(* Calculates the size of this message in Protocol Buffer wire format, in bytes. *)
METHOD CalculateSize : UDINT
VAR
    nSize : UDINT;
    nRepeatedFieldSize : UDINT;
END_VAR
// repeated EnumOfTypeSint enum_values_sint = 1;
_fbRepeatedId1.CalculateSize(nSize => nRepeatedFieldSize);
nSize := nSize + nRepeatedFieldSize;
CalculateSize := nSize;
END_METHOD

(* Merges the data from the specified coded input stream with the current message.*)
METHOD MergeFrom : HRESULT
VAR_IN_OUT
    fbParseCtx : FB_ParseContext;
END_VAR
VAR
    nTag : UDINT;
END_VAR
_fbRepeatedId1.Initialize();
REPEAT
MergeFrom := fbParseCtx.ReadTag(nTag=> nTag);
IF SUCCEEDED(MergeFrom) AND nTag = 0 THEN
    EXIT;
END_IF;

IF FAILED(MergeFrom) THEN
    RETURN;
END_IF

CASE nTag OF
    16#0A:    // repeated EnumOfTypeSint enum_values_sint = 1;
        MergeFrom := _fbRepeatedId1.AddEntriesFrom(fbParseCtx:= fbParseCtx, ipFieldCodec:= _fbFieldCodecId1,nCount=> _stRepeatedEnumTests.enum_values_sint_count);
ELSE
    MergeFrom := fbParseCtx.SkipLastField();
END_CASE

UNTIL (FAILED(MergeFrom) OR nTag = 0)
END_REPEAT
END_METHOD

PROPERTY PUBLIC MessageValue : T_Any
GET
MessageValue := F_ToAnyType(anyArg:= _stRepeatedEnumTests);
END_GET
END_PROPERTY

PROPERTY PUBLIC Parser : REFERENCE TO FB_MessageParser
GET
Parser REF= THIS^._fbMessageParser;
END_GET
END_PROPERTY

PROPERTY PUBLIC RepeatedEnumTests : ST_RepeatedEnumTests
GET
RepeatedEnumTests := _stRepeatedEnumTests;
END_GET
SET
_stRepeatedEnumTests := RepeatedEnumTests;
END_SET
END_PROPERTY

(* Writer for this message.*)
PROPERTY PUBLIC Writer : REFERENCE TO FB_MessageWriter
GET
Writer REF= THIS^._fbMessageWriter;
END_GET
END_PROPERTY

(* Writes the data to the given coded output stream.*)
METHOD WriteTo : HRESULT
VAR_IN_OUT
	(* Coded output stream to write the data to. *)
	fbWriteCtx	: FB_WriteContext;
END_VAR
// repeated EnumOfTypeSint enum_values_sint = 1;
WriteTo := _fbRepeatedId1.WriteToWithCount(fbWriteCtx:= fbWriteCtx, ipFieldCodec:= _fbFieldCodecId1, nCount:= _stRepeatedEnumTests.enum_values_sint_count);
IF FAILED(WriteTo) THEN
    RETURN;
END_IF
END_METHOD

END_FUNCTION_BLOCK

// ---- FieldCodec/FB_FieldCodecFloat.TcPOU
FUNCTION_BLOCK FB_FieldCodecFloat EXTENDS FB_FieldCodec
VAR_INPUT
END_VAR
VAR_OUTPUT
END_VAR
VAR
    fValue : REAL;
END_VAR

METHOD CalculatePackedDataSize : HRESULT
VAR_INPUT CONSTANT
	anyFirstElem	: T_Any;
	nLength	        : UDINT;        // items to write
END_VAR
VAR_OUTPUT
    nPackedDataSize : UDINT;
END_VAR
VAR
    anyItem         : T_ANY;
    i               : UDINT;
    fValue          : REAL;
END_VAR
anyItem := anyFirstElem;

IF nLength < 1 THEN
    nPackedDataSize := 0;
    RETURN;
END_IF

FOR i := 0  TO nLength - 1 DO
    anyItem.pValue := anyFirstElem.pValue + (i * TO_UDINT(anyFirstElem.diSize)); 
    fValue := PREAL_TO_REAL(anyItem.pValue);
    nPackedDataSize := nPackedDataSize + F_ComputeFloatSize(fValue);
END_FOR
END_METHOD

METHOD IsPackedRepeatedField : BOOL
VAR_INPUT
	nTag	: UDINT;
END_VAR
IsPackedRepeatedField := F_IsPackedRepeatedField(nTag);
END_METHOD


METHOD ValueReader : HRESULT
VAR_IN_OUT      
    stCtx : ST_ParseContext;
END_VAR
VAR_OUTPUT
	anyOut	: T_Any;
END_VAR

ValueReader := F_ParseFloat(stCtx, fValue=> fValue);
anyOut := F_ToAnyType(anyArg:= fValue);
END_METHOD

METHOD ValueWriter : HRESULT
VAR_IN_OUT
    stCtx  : ST_WriteContext;
END_VAR
VAR_INPUT
    anyIn : T_ANY;
END_VAR
VAR
    fValue  : REAL;
END_VAR

fValue := PREAL_TO_REAL(anyIn.pValue);
ValueWriter := F_WriteFloat(stCtx, fValue);
END_METHOD

END_FUNCTION_BLOCK

// ---- FieldCodec/FB_FieldCodecSint32.TcPOU
FUNCTION_BLOCK FB_FieldCodecSint32 EXTENDS FB_FieldCodec
VAR_INPUT
END_VAR
VAR_OUTPUT
END_VAR
VAR
    nValue : DINT;
END_VAR

METHOD CalculatePackedDataSize : HRESULT
VAR_INPUT CONSTANT
	anyFirstElem	: T_Any;
	nLength	        : UDINT;        // items to write
END_VAR
VAR_OUTPUT
    nPackedDataSize : UDINT;
END_VAR
VAR
    anyItem         : T_ANY;
    i               : UDINT;
    nValue          : DINT;
END_VAR
anyItem := anyFirstElem;

IF nLength < 1 THEN
    nPackedDataSize := 0;
    RETURN;
END_IF

FOR i := 0  TO nLength - 1 DO
    anyItem.pValue := anyFirstElem.pValue + (i * TO_UDINT(anyFirstElem.diSize)); 
    nValue := PDINT_TO_DINT(anyItem.pValue);
    nPackedDataSize := nPackedDataSize + F_ComputeSInt32Size(nValue);
END_FOR
END_METHOD

METHOD IsPackedRepeatedField : BOOL
VAR_INPUT
	nTag	: UDINT;
END_VAR
IsPackedRepeatedField := F_IsPackedRepeatedField(nTag);
END_METHOD


METHOD ValueReader : HRESULT
VAR_IN_OUT      
    stCtx : ST_ParseContext;
END_VAR
VAR_OUTPUT
	anyOut	: T_Any;
END_VAR
VAR
    nTmp : UDINT;
END_VAR

ValueReader := F_ParseRawVarint32(stCtx, nTmp);
IF FAILED(ValueReader) THEN
    RETURN;
END_IF
nValue := F_DecodeZigZag32(nTmp);
anyOut := F_ToAnyType(anyArg:= nValue);
END_METHOD

METHOD ValueWriter : HRESULT
VAR_IN_OUT
    stCtx  : ST_WriteContext;
END_VAR
VAR_INPUT
    anyIn : T_ANY;
END_VAR
VAR
    nValue  : DINT;
END_VAR

nValue := PDINT_TO_DINT(anyIn.pValue);
ValueWriter := F_WriteSInt32(stCtx, nValue);
END_METHOD

END_FUNCTION_BLOCK

// ---- FieldCodec/FB_FieldCodecInt64.TcPOU
FUNCTION_BLOCK FB_FieldCodecInt64 EXTENDS FB_FieldCodec
VAR_INPUT
END_VAR
VAR_OUTPUT
END_VAR
VAR
    nValue : ULINT;
END_VAR

METHOD CalculatePackedDataSize : HRESULT
VAR_INPUT CONSTANT
	anyFirstElem	: T_Any;
	nLength	        : UDINT;        // items to write
END_VAR
VAR_OUTPUT
    nPackedDataSize : UDINT;
END_VAR
VAR
    anyItem         : T_ANY;
    i               : UDINT;
    nValue          : LINT;
END_VAR
anyItem := anyFirstElem;

IF nLength < 1 THEN
    nPackedDataSize := 0;
    RETURN;
END_IF

FOR i := 0  TO nLength - 1 DO
    anyItem.pValue := anyFirstElem.pValue + (i * TO_UDINT(anyFirstElem.diSize)); 
    nValue := PLINT_TO_LINT(anyItem.pValue);
    nPackedDataSize := nPackedDataSize + F_ComputeInt64Size(nValue);
END_FOR
END_METHOD

METHOD IsPackedRepeatedField : BOOL
VAR_INPUT
	nTag	: UDINT;
END_VAR
IsPackedRepeatedField := F_IsPackedRepeatedField(nTag);
END_METHOD


METHOD ValueReader : HRESULT
VAR_IN_OUT      
    stCtx : ST_ParseContext;
END_VAR
VAR_OUTPUT
	anyOut	: T_Any;
END_VAR

ValueReader := F_ParseRawVarint64(stCtx, nValue);
anyOut := F_ToAnyType(anyArg:= nValue);
END_METHOD

METHOD ValueWriter : HRESULT
VAR_IN_OUT
    stCtx  : ST_WriteContext;
END_VAR
VAR_INPUT
    anyIn : T_ANY;
END_VAR
VAR
    nValue  : LINT;
END_VAR

nValue := PLINT_TO_LINT(anyIn.pValue);
ValueWriter := F_WriteInt64(stCtx, nValue);
END_METHOD

END_FUNCTION_BLOCK

// ---- FieldCodec/FB_FieldCodecSint64.TcPOU
FUNCTION_BLOCK FB_FieldCodecSint64 EXTENDS FB_FieldCodec
VAR_INPUT
END_VAR
VAR_OUTPUT
END_VAR
VAR
    nValue : LINT;
END_VAR

METHOD CalculatePackedDataSize : HRESULT
VAR_INPUT CONSTANT
	anyFirstElem	: T_Any;
	nLength	        : UDINT;        // items to write
END_VAR
VAR_OUTPUT
    nPackedDataSize : UDINT;
END_VAR
VAR
    anyItem         : T_ANY;
    i               : UDINT;
    nValue          : LINT;
END_VAR
anyItem := anyFirstElem;

IF nLength < 1 THEN
    nPackedDataSize := 0;
    RETURN;
END_IF

FOR i := 0  TO nLength - 1 DO
    anyItem.pValue := anyFirstElem.pValue + (i * TO_UDINT(anyFirstElem.diSize)); 
    nValue := PLINT_TO_LINT(anyItem.pValue);
    nPackedDataSize := nPackedDataSize + F_ComputeSInt64Size(nValue);
END_FOR
END_METHOD

METHOD IsPackedRepeatedField : BOOL
VAR_INPUT
	nTag	: UDINT;
END_VAR
IsPackedRepeatedField := F_IsPackedRepeatedField(nTag);
END_METHOD


METHOD ValueReader : HRESULT
VAR_IN_OUT      
    stCtx : ST_ParseContext;
END_VAR
VAR_OUTPUT
	anyOut	: T_Any;
END_VAR
VAR 
    nTmp : ULINT;
END_VAR

ValueReader := F_ParseRawVarint64(stCtx, nTmp);
IF FAILED(ValueReader) THEN
    RETURN;
END_IF
nValue := F_DecodeZigZag64(nTmp);
anyOut := F_ToAnyType(anyArg:= nValue);
END_METHOD

METHOD ValueWriter : HRESULT
VAR_IN_OUT
    stCtx  : ST_WriteContext;
END_VAR
VAR_INPUT
    anyIn : T_ANY;
END_VAR
VAR
    nValue  : LINT;
END_VAR

nValue := PLINT_TO_LINT(anyIn.pValue);
ValueWriter := F_WriteSInt64(stCtx, nValue);
END_METHOD

END_FUNCTION_BLOCK

// ---- Helper/POUs/F_ToAnyBit.TcPOU
FUNCTION F_ToAnyBit : T_AnyBit
VAR_INPUT
    anyBit	: ANY_BIT;
END_VAR

F_ToAnyBit := anyBit;

END_FUNCTION

// ---- Helper/POUs/F_ToAnyInt.TcPOU
FUNCTION F_ToAnyInt : T_AnyInt
VAR_INPUT
    anyInt	: ANY_INT;
END_VAR

F_ToAnyInt := anyInt;

END_FUNCTION

// ---- Helper/POUs/F_ToAnyNum.TcPOU
FUNCTION F_ToAnyNum : T_AnyNum
VAR_INPUT
    anyNum	: ANY_NUM;
END_VAR

F_ToAnyNum := anyNum;

END_FUNCTION

// ---- ParsingPrimitives/POUs/F_ReadStringInternal.TcPOU
// Reads a string field value from the input.
FUNCTION INTERNAL F_ReadStringInternal : HRESULT
VAR_IN_OUT      
    stCtx : ST_ParseContext;
END_VAR
VAR_INPUT
    stAnyStringOut : T_Any;   
END_VAR
VAR
    nStrLength : UDINT;
END_VAR

F_ReadStringInternal := S_OK;

F_ReadStringInternal := F_ParseLength(stCtx, nLength=> nStrLength);
IF FAILED(F_ReadStringInternal) THEN
    RETURN;
END_IF

F_ReadStringInternal := F_ReadRawString(stCtx, nStrLength, stAnyStringOut);

END_FUNCTION

// ---- POUs/ComputeSize/F_ComputeTagSize.TcPOU
FUNCTION F_ComputeTagSize : UDINT
VAR_INPUT
    nFieldnumber    : UDINT;
END_VAR


F_ComputeTagSize := F_ComputeRawVarint32Size(nValue:= F_MakeTag(nFieldNumber, 0));

END_FUNCTION

// ---- Project Information/F_GetCompany.TcPOU
// This function has been automatically generated from the project information.
{attribute 'signature_flag' := '1073741824'}
{attribute 'TcGenerated'}
{attribute 'no-analysis'}
FUNCTION F_GetCompany : WSTRING
VAR_INPUT
	
END_VAR

F_GetCompany := "TcHaxx";

END_FUNCTION

// ---- Project Information/F_GetTitle.TcPOU
// This function has been automatically generated from the project information.
{attribute 'signature_flag' := '1073741824'}
{attribute 'TcGenerated'}
{attribute 'no-analysis'}
FUNCTION F_GetTitle : WSTRING
VAR_INPUT
	
END_VAR

F_GetTitle := "protobuf";

END_FUNCTION

// ---- Project Information/F_GetVersion.TcPOU
// This function has been automatically generated from the project information.
{attribute 'signature_flag' := '1073741824'}
{attribute 'TcGenerated'}
{attribute 'no-analysis'}
FUNCTION F_GetVersion : ST_LibVersion
VAR_INPUT
	
END_VAR

F_GetVersion.iMajor := 0;
F_GetVersion.iMinor := 0;
F_GetVersion.iBuild := 1;
F_GetVersion.iRevision := 0;
F_GetVersion.sVersion := '0.0.1.0';
F_GetVersion.nFlags := 0;

END_FUNCTION

// ---- WritingPrimitives/POUs/F_WriteRawLittleEndian32.TcPOU
// Writes a 32-bit little-endian integer.
FUNCTION F_WriteRawLittleEndian32 : HRESULT
VAR_IN_OUT      
    stCtx : ST_WriteContext;
END_VAR
VAR_INPUT CONSTANT
    nValue : UDINT;
END_VAR
VAR CONSTANT
    cLength : UDINT := SIZEOF(nValue);
END_VAR

F_WriteRawLittleEndian32 := F_WriteToBuffer(stCtx, F_ToAnyType(nValue), cLength);

END_FUNCTION

// ---- WritingPrimitives/POUs/F_WriteRawLittleEndian64.TcPOU
// Writes a 64-bit little-endian integer.
FUNCTION F_WriteRawLittleEndian64 : HRESULT
VAR_IN_OUT      
    stCtx : ST_WriteContext;
END_VAR
VAR_INPUT CONSTANT
    nValue : ULINT;
END_VAR
VAR CONSTANT
    cLength : UDINT := SIZEOF(nValue);
END_VAR

F_WriteRawLittleEndian64 := F_WriteToBuffer(stCtx, F_ToAnyType(nValue), cLength);

END_FUNCTION

// ---- __TESTs/EnumTests/FB_ReadEnumTests.TcPOU
FUNCTION_BLOCK INTERNAL FINAL FB_ReadEnumTests EXTENDS FB_TestSuite
VAR_INPUT
END_VAR
VAR_OUTPUT
END_VAR
VAR
	eActual : (UNINITIALIZED:= 16#ABAB) := UNINITIALIZED;
	eExpected : ARRAY[0..2] OF (NEG255:= -255, POS255:= 255, ZERO:= 0);
END_VAR

FailsWithInvalidDataForNonEnumType();
ShouldReadEnumValueTheory();

METHOD PRIVATE FailsWithInvalidDataForNonEnumType : BOOL
VAR_INPUT
END_VAR
VAR_INST
	fbSut	: FB_ParseContext;
END_VAR
VAR
	aBuffer	: ARRAY[0..15] OF BYTE := [16#80, 16#01];
	hr : HRESULT;
	nNonEnumVar	: DINT;
END_VAR
VAR CONSTANT
	cHrExpected : HRESULT := E_HRESULTAdsErr.INVALIDDATA;
END_VAR
TEST(__POUNAME());

//Arrange
fbSut.FromBuffer(aBuffer);

// Act
hr := fbSut.ReadEnum(anyEnum:= nNonEnumVar);

//Assert
AssertEquals_DINT(
    Expected:= cHrExpected,
    Actual:= hr,
    Message:= CONCAT(CONCAT('Expected ', TO_STRING(cHrExpected)), ' for non Enum.'));

AssertEquals_UDINT(
	Expected:= 0,
	Actual:= fbSut.refCtx.stState.nBufferPos,
	Message:= 'Unexpected change to ParseContext buffer position.');

TEST_FINISHED_NAMED(__POUNAME());
END_METHOD

METHOD PRIVATE ShouldReadEnumValue : BOOL
// VAR_IN_OUT CONSTANT
// 	aBuffer : ARRAY[*] OF BYTE;
// END_VAR
VAR_INPUT
	nEnumValueBuffer : DINT;
	nExpected : INT;
END_VAR
VAR_INST
    fbSut : FB_ParseContext;
	fbWrCtx : FB_WriteContext;
END_VAR
VAR
	hr : HRESULT;
	aBuffer : ARRAY[0..31] OF BYTE;
END_VAR
// Arrange
fbSut.FromBuffer(aBuffer);
fbWrCtx.FromBuffer(aBuffer);
F_WriteInt32(fbWrCtx.refCtx, nValue:= nEnumValueBuffer);
eActual := UNINITIALIZED;
eExpected[0] := UNINITIALIZED;	// neighbour guard
eExpected[1] := nExpected;
eExpected[2] := UNINITIALIZED;  // neighbour guard

// Act
hr := fbSut.ReadEnum(anyEnum:= eActual);

//Assert
AssertEquals_DINT(Expected:= S_OK, Actual:= hr, Message:= 'Failed to read enum value.');
AssertEquals_INT(Expected:= eExpected[0], Actual:= UNINITIALIZED, Message:= 'Lower neighbor value was unexpectedly modified.');
AssertEquals_INT(Expected:= eExpected[1], Actual:= eActual, Message:= '');
AssertEquals_INT(Expected:= eExpected[2], Actual:= UNINITIALIZED, Message:= 'Upper neighbor value was unexpectedly modified.');
END_METHOD

METHOD PRIVATE ShouldReadEnumValueTheory : BOOL
VAR_INPUT
END_VAR
TEST(__POUNAME());
ShouldReadEnumValue(nEnumValueBuffer:= 0, nExpected:= ZERO);
ShouldReadEnumValue(nEnumValueBuffer:= POS255, nExpected:= POS255);
ShouldReadEnumValue(nEnumValueBuffer:= 257, nExpected:= 257);
ShouldReadEnumValue(nEnumValueBuffer:= NEG255, nExpected:= NEG255);
ShouldReadEnumValue(nEnumValueBuffer:= 32767, nExpected:= 32767);
ShouldReadEnumValue(nEnumValueBuffer:= -32768, nExpected:= -32768);
ShouldReadEnumValue(nEnumValueBuffer:= 65535, nExpected:= -1);  // 16#0000_FFFF --> -1 (INT)
ShouldReadEnumValue(nEnumValueBuffer:= 65536, nExpected:= 0);  // 16#0001_0000 --> 0 (INT)
ShouldReadEnumValue(nEnumValueBuffer:= -65535, nExpected:= 1);  // 16#FFFF_0001 --> 16#0001 (INT)
ShouldReadEnumValue(nEnumValueBuffer:= 65409, nExpected:= -127);
TEST_FINISHED_NAMED(__POUNAME());
END_METHOD

END_FUNCTION_BLOCK

// ---- __TESTs/EnumTests/FB_WriteEnumTests.TcPOU
FUNCTION_BLOCK INTERNAL FINAL FB_WriteEnumTests EXTENDS FB_TestSuite
VAR_INPUT
END_VAR
VAR_OUTPUT
END_VAR
VAR
	eActual : (UNINITIALIZED:= 16#ABAB) := UNINITIALIZED;
END_VAR

FailsWithInvalidDataForNonEnumType();
ShouldWriteEnumValueTheory();

METHOD PRIVATE FailsWithInvalidDataForNonEnumType : BOOL
VAR_INPUT
END_VAR
VAR_INST
	fbSut	: FB_WriteContext;
END_VAR
VAR
	aBuffer	: ARRAY[0..15] OF BYTE;
	hr : HRESULT;
	nNonEnumVar	: DINT;
END_VAR
VAR CONSTANT
	cHrExpected : HRESULT := E_HRESULTAdsErr.INVALIDDATA;
END_VAR
TEST(__POUNAME());

//Arrange
fbSut.FromBuffer(aBuffer);

// Act
hr := fbSut.WriteEnum(anyEnum:= nNonEnumVar);

//Assert
AssertEquals_DINT(
    Expected:= cHrExpected,
    Actual:= hr,
    Message:= CONCAT(CONCAT('Expected ', TO_STRING(cHrExpected)), ' for non Enum.'));

AssertEquals_UDINT(
	Expected:= 0,
	Actual:= fbSut.refCtx.stState.nBufferPos,
	Message:= 'Unexpected change to ParseContext buffer position.');

TEST_FINISHED_NAMED(__POUNAME());
END_METHOD

METHOD PRIVATE ShouldWriteEnumValue : BOOL
VAR_IN_OUT CONSTANT
    aExpectedBuffer     : ARRAY [*] OF BYTE;    
END_VAR
VAR_INPUT
	nEnumValue : INT;
	nExpectedBufferPos  : UDINT;
END_VAR
VAR_INST
	fbSut : FB_WriteContext;
END_VAR
VAR
	hr : HRESULT;
	aActualBuffer : ARRAY[0..31] OF BYTE;
END_VAR
// Arrange
fbSut.FromBuffer(aActualBuffer);
eActual := nEnumValue;

// Act
hr := fbSut.WriteEnum(anyEnum:= eActual);

// Assert
AssertEquals_DINT(
     Expected:= S_OK,
     Actual:= hr,
     Message:= 'Expected S_OK instead of error');

{warning disable C0041}
AssertArrayEquals_BYTE(    
    Expecteds:= aExpectedBuffer,
    Actuals:= aActualBuffer,
    MEssage:= CONCAT('Expected buffers to be equal for Enum value ', TO_STRING(nEnumValue))
);

AssertEquals_UDINT(
    Expected:= nExpectedBufferPos,
    Actual:= fbSut.refCtx.stState.nBufferPos,
    Message:= CONCAT(CONCAT('Expected stState.nBufferPos to equal ', TO_STRING(nExpectedBufferPos)), CONCAT(', for Enum value ', TO_STRING(nExpectedBufferPos))));
END_METHOD

METHOD PRIVATE ShouldWriteEnumValueTheory : BOOL
VAR CONSTANT
	aBufferZero : ARRAY[0..31] OF BYTE := [];
	aBufferOne :  ARRAY[0..31] OF BYTE := [16#01];
	aBufferValue127 : ARRAY[0..31] OF BYTE := [16#7F];
	aBufferValueNeg127 : ARRAY[0..31] OF BYTE := [16#81, 16#FF, 16#03];
	aBufferValueNeg32768 : ARRAY[0..31] OF BYTE := [16#80, 16#80, 16#02];
	aBufferValue32767 : ARRAY[0..31] OF BYTE := [16#FF, 16#FF, 16#01];
END_VAR
TEST(__POUNAME());
ShouldWriteEnumValue(aExpectedBuffer:= aBufferZero, nEnumValue:= 0, nExpectedBufferPos:= 1);
ShouldWriteEnumValue(aExpectedBuffer:= aBufferOne, nEnumValue:= 1, nExpectedBufferPos:= 1);
ShouldWriteEnumValue(aExpectedBuffer:= aBufferValue127, nEnumValue:= 127, nExpectedBufferPos:= 1);
ShouldWriteEnumValue(aExpectedBuffer:= aBufferValueNeg127, nEnumValue:= -127, nExpectedBufferPos:= 3);
ShouldWriteEnumValue(aExpectedBuffer:= aBufferValueNeg32768, nEnumValue:= -32768, nExpectedBufferPos:= 3);
ShouldWriteEnumValue(aExpectedBuffer:= aBufferValue32767, nEnumValue:= 32767, nExpectedBufferPos:= 3);
TEST_FINISHED_NAMED(__POUNAME());
END_METHOD

END_FUNCTION_BLOCK

// ---- __TESTs/RepeatedFieldTests/Write/FB_WriteRepeatedFieldDoubleTests.TcPOU
FUNCTION_BLOCK INTERNAL FINAL FB_WriteRepeatedFieldDoubleTests EXTENDS FB_TestSuite
VAR_INPUT
END_VAR
VAR_OUTPUT
END_VAR
VAR
    fbFieldCodec : FB_FieldCodecDouble(nTag:= 0);
	aActual    	 : ARRAY [0..7] OF LREAL;
	fbRepeatedField		: FB_RepeatedField(anyArray:= F_ToAnyType(aActual), anyFirstElem:= F_ToAnyType(aActual[0]), ipFieldCodec:= fbFieldCodec);
END_VAR

ShouldWriteRepeatedFieldTheory();

METHOD PRIVATE Reset
VAR_INPUT
END_VAR
fbRepeatedField.Initialize();
MEMSET(destAddr:= ADR(aActual), fillByte:= 16#0, n:= SIZEOF(aActual));
END_METHOD

METHOD PRIVATE ShouldWriteRepeatedField
VAR_IN_OUT CONSTANT
    aExpected   : ARRAY [*] OF BYTE;
END_VAR
VAR_INPUT
    aValues     : ARRAY [0..7] OF LREAL;
    nLength     : UDINT;
    nTag        : UDINT;
    nBufferPosStart     : UDINT;
    nExpectedBufferPos  : UDINT;
    ipFieldCodec        : I_FieldCodec;
END_VAR
VAR_INST
    fbCtx   : FB_WriteContext;
END_VAR
VAR
    aActualBuffer       : ARRAY [0..63] OF BYTE;
    hr                  : HRESULT;

END_VAR
// Arrange
Reset();
fbCtx.FromBuffer(aActualBuffer);
fbCtx.refCtx.stState.nBufferPos := nBufferPosStart;
ipFieldCodec.Tag := nTag;
fbRepeatedField.InitializeFromArray(anyArray:= F_ToAnyType(aValues), anyFirstElem:= F_ToAnyType(aValues[0]), nCount:= nLength);

// Act
hr := fbRepeatedField.WriteTo(fbWriteCtx:= fbCtx, ipFieldCodec:= ipFieldCodec);

// Assert
AssertEquals_DINT(
    Expected:= S_OK,
    Actual:= hr,
    Message:= 'Expected S_OK instead of error');
    
{warning disable C0041}
AssertArrayEquals_BYTE(Expecteds:= aExpected, Actuals:= aActualBuffer, Message:= '');
 
AssertEquals_UDINT(
    Expected:= nExpectedBufferPos,
    Actual:= fbCtx.refCtx.stState.nBufferPos,
    Message:= CONCAT('Expected stState.nBufferPos to equal ', TO_STRING(nExpectedBufferPos)));
END_METHOD

METHOD PRIVATE ShouldWriteRepeatedFieldTheory : REFERENCE TO FB_Test
VAR CONSTANT
    cRawValueZeroLength     : ARRAY[0..63] OF BYTE := [16#00, 16#00];
    cRawValue1              : ARRAY[0..63] OF BYTE := [16#00, 16#22, 16#30, 16#00, 16#00, 16#00, 16#00, 16#00, 16#00, 16#00, 16#00, 16#54, 16#E3, 16#A5, 16#9B, 16#44, 16#4A, 16#93, 16#40, 16#E7, 16#1D, 16#A7, 16#E8, 16#88, 16#E4, 16#94, 16#40, 16#00, 16#00, 16#00, 16#00, 16#00, 16#00, 16#F0, 16#BF, 16#A2, 16#5B, 16#F3, 16#C3, 16#29, 16#8C, 16#67, 16#41, 16#DD, 16#9A, 16#9F, 16#06, 16#00, 16#00, 16#E0, 16#41];  
END_VAR

VAR CONSTANT
    aExpectedZeroLength     : ARRAY [0..7] OF LREAL := [0, 0, 0, 0, 0, 0, 0, 0];
    aExpected1              : ARRAY [0..7] OF LREAL := [0, 1234.567, 1337.1337, -1.0, 12345678.12345678, 2147483700.987654];
END_VAR
TEST(__POUNAME());

ShouldWriteRepeatedField(aExpected:= cRawValueZeroLength, aValues:= aExpectedZeroLength, nLength:= 0, nTag:= F_MakeTag(1, E_WireType.LengthDelimited), nBufferPosStart:= 0, nExpectedBufferPos:= 0, ipFieldCodec:= THIS^.fbFieldCodec);
ShouldWriteRepeatedField(aExpected:= cRawValue1, aValues:= aExpected1, nLength:= 6, nTag:= F_MakeTag(4, E_WireType.LengthDelimited), nBufferPosStart:= 1, nExpectedBufferPos:= 51, ipFieldCodec:= THIS^.fbFieldCodec);

TEST_FINISHED_NAMED(__POUNAME());
END_METHOD

END_FUNCTION_BLOCK

// ---- __TESTs/RepeatedFieldTests/Write/FB_WriteRepeatedFieldFixed32Tests.TcPOU
FUNCTION_BLOCK INTERNAL FINAL FB_WriteRepeatedFieldFixed32Tests EXTENDS FB_TestSuite
VAR_INPUT
END_VAR
VAR_OUTPUT
END_VAR
VAR
    fbFieldCodec : FB_FieldCodecFixed32(nTag:= 0);
	aActual     : ARRAY [0..7] OF DINT;
	fbRepeatedField		: FB_RepeatedField(anyArray:= F_ToAnyType(aActual), anyFirstElem:= F_ToAnyType(aActual[0]), ipFieldCodec:= fbFieldCodec);
END_VAR

ShouldWriteRepeatedFieldTheory();

METHOD PRIVATE Reset
VAR_INPUT
END_VAR
fbRepeatedField.Initialize();
MEMSET(destAddr:= ADR(aActual), fillByte:= 16#0, n:= SIZEOF(aActual));
END_METHOD

METHOD PRIVATE ShouldWriteRepeatedField
VAR_IN_OUT CONSTANT
    aExpected   : ARRAY [*] OF BYTE;
END_VAR
VAR_INPUT
    aValues     : ARRAY [0..7] OF DINT;
    nLength     : UDINT;
    nTag        : UDINT;
    nBufferPosStart     : UDINT;
    nExpectedBufferPos  : UDINT;
    ipFieldCodec        : I_FieldCodec;
END_VAR
VAR_INST
    fbCtx   : FB_WriteContext;
END_VAR
VAR
    aActualBuffer       : ARRAY [0..63] OF BYTE;
    hr                  : HRESULT;

END_VAR
// Arrange
Reset();
fbCtx.FromBuffer(aActualBuffer);
fbCtx.refCtx.stState.nBufferPos := nBufferPosStart;
ipFieldCodec.Tag := nTag;
fbRepeatedField.InitializeFromArray(anyArray:= F_ToAnyType(aValues), anyFirstElem:= F_ToAnyType(aValues[0]), nCount:= nLength);

// Act
hr := fbRepeatedField.WriteTo(fbWriteCtx:= fbCtx, ipFieldCodec:= ipFieldCodec);

// Assert
AssertEquals_DINT(
    Expected:= S_OK,
    Actual:= hr,
    Message:= 'Expected S_OK instead of error');
    
{warning disable C0041}
AssertArrayEquals_BYTE(Expecteds:= aExpected, Actuals:= aActualBuffer, Message:= '');
 
AssertEquals_UDINT(
    Expected:= nExpectedBufferPos,
    Actual:= fbCtx.refCtx.stState.nBufferPos,
    Message:= CONCAT('Expected stState.nBufferPos to equal ', TO_STRING(nExpectedBufferPos)));
END_METHOD

METHOD PRIVATE ShouldWriteRepeatedFieldTheory : REFERENCE TO FB_Test
VAR CONSTANT
    cRawValueZeroLength     : ARRAY[0..63] OF BYTE := [16#00, 16#00];
    cRawValue1              : ARRAY[0..63] OF BYTE := [16#00, 16#0A, 16#18, 16#00, 16#00, 16#00, 16#00, 16#D2, 16#04, 16#00, 16#00, 16#39, 16#05, 16#00, 16#00, 16#FF, 16#FF, 16#FF, 16#FF, 16#4E, 16#61, 16#BC, 16#00, 16#FF, 16#FF, 16#FF, 16#7F];  
END_VAR

VAR CONSTANT
    aExpectedZeroLength     : ARRAY [0..7] OF DINT := [0, 0, 0, 0, 0, 0, 0, 0];
    aExpected1              : ARRAY [0..7] OF DINT := [0, 1234, 1337, -1, 12345678, 2147483647];
END_VAR
TEST(__POUNAME());

ShouldWriteRepeatedField(aExpected:= cRawValueZeroLength, aValues:= aExpectedZeroLength, nLength:= 0, nTag:= F_MakeTag(1, E_WireType.LengthDelimited), nBufferPosStart:= 0, nExpectedBufferPos:= 0, ipFieldCodec:= THIS^.fbFieldCodec);
ShouldWriteRepeatedField(aExpected:= cRawValue1, aValues:= aExpected1, nLength:= 6, nTag:= F_MakeTag(1, E_WireType.LengthDelimited), nBufferPosStart:= 1, nExpectedBufferPos:= 27, ipFieldCodec:= THIS^.fbFieldCodec);

TEST_FINISHED_NAMED(__POUNAME());
END_METHOD

END_FUNCTION_BLOCK

// ---- __TESTs/RepeatedFieldTests/Write/FB_WriteRepeatedFieldFixed64Tests.TcPOU
FUNCTION_BLOCK INTERNAL FINAL FB_WriteRepeatedFieldFixed64Tests EXTENDS FB_TestSuite
VAR_INPUT
END_VAR
VAR_OUTPUT
END_VAR
VAR
	fbFieldCodec : FB_FieldCodecFixed64(nTag:= 0);
	aActual    	 : ARRAY [0..7] OF LINT;
	fbRepeatedField		: FB_RepeatedField(anyArray:= F_ToAnyType(aActual), anyFirstElem:= F_ToAnyType(aActual[0]), ipFieldCodec:= fbFieldCodec);
END_VAR

ShouldWriteRepeatedFieldTheory();

METHOD PRIVATE Reset
VAR_INPUT
END_VAR
fbRepeatedField.Initialize();
MEMSET(destAddr:= ADR(aActual), fillByte:= 16#0, n:= SIZEOF(aActual));
END_METHOD

METHOD PRIVATE ShouldWriteRepeatedField
VAR_IN_OUT CONSTANT
    aExpected   : ARRAY [*] OF BYTE;
END_VAR
VAR_INPUT
    aValues     : ARRAY [0..7] OF LINT;
    nLength     : UDINT;
    nTag        : UDINT;
    nBufferPosStart     : UDINT;
    nExpectedBufferPos  : UDINT;
    ipFieldCodec        : I_FieldCodec;
END_VAR
VAR_INST
    fbCtx   : FB_WriteContext;
END_VAR
VAR
    aActualBuffer       : ARRAY [0..63] OF BYTE;
    hr                  : HRESULT;

END_VAR
// Arrange
Reset();
fbCtx.FromBuffer(aActualBuffer);
fbCtx.refCtx.stState.nBufferPos := nBufferPosStart;
ipFieldCodec.Tag := nTag;
fbRepeatedField.InitializeFromArray(anyArray:= F_ToAnyType(aValues), anyFirstElem:= F_ToAnyType(aValues[0]), nCount:= nLength);

// Act
hr := fbRepeatedField.WriteTo(fbWriteCtx:= fbCtx, ipFieldCodec:= ipFieldCodec);

// Assert
AssertEquals_DINT(
    Expected:= S_OK,
    Actual:= hr,
    Message:= 'Expected S_OK instead of error');
    
{warning disable C0041}
AssertArrayEquals_BYTE(Expecteds:= aExpected, Actuals:= aActualBuffer, Message:= '');
 
AssertEquals_UDINT(
    Expected:= nExpectedBufferPos,
    Actual:= fbCtx.refCtx.stState.nBufferPos,
    Message:= CONCAT('Expected stState.nBufferPos to equal ', TO_STRING(nExpectedBufferPos)));
END_METHOD

METHOD PRIVATE ShouldWriteRepeatedFieldTheory : REFERENCE TO FB_Test
VAR CONSTANT
    cRawValueZeroLength     : ARRAY[0..63] OF BYTE := [16#00, 16#00];
    cRawValue1              : ARRAY[0..63] OF BYTE := [16#00, 16#0A, 16#30, 16#00, 16#00, 16#00, 16#00, 16#00, 16#00, 16#00, 16#00, 16#D2, 16#04, 16#00, 16#00, 16#00, 16#00, 16#00, 16#00, 16#39, 16#05, 16#00, 16#00, 16#00, 16#00, 16#00, 16#00, 16#FF, 16#FF, 16#FF, 16#FF, 16#FF, 16#FF, 16#FF, 16#FF, 16#4E, 16#61, 16#BC, 16#00, 16#00, 16#00, 16#00, 16#00, 16#34, 16#00, 16#00, 16#80, 16#00, 16#00, 16#00, 16#00];  
END_VAR

VAR CONSTANT
    aExpectedZeroLength     : ARRAY [0..7] OF LINT := [0, 0, 0, 0, 0, 0, 0, 0];
    aExpected1              : ARRAY [0..7] OF LINT := [0, 1234, 1337, -1, 12345678, 2147483700];
END_VAR
TEST(__POUNAME());

ShouldWriteRepeatedField(aExpected:= cRawValueZeroLength, aValues:= aExpectedZeroLength, nLength:= 0, nTag:= F_MakeTag(1, E_WireType.LengthDelimited), nBufferPosStart:= 0, nExpectedBufferPos:= 0, ipFieldCodec:= THIS^.fbFieldCodec);
ShouldWriteRepeatedField(aExpected:= cRawValue1, aValues:= aExpected1, nLength:= 6, nTag:= F_MakeTag(1, E_WireType.LengthDelimited), nBufferPosStart:= 1, nExpectedBufferPos:= 51, ipFieldCodec:= THIS^.fbFieldCodec);

TEST_FINISHED_NAMED(__POUNAME());
END_METHOD

END_FUNCTION_BLOCK

// ---- __TESTs/RepeatedFieldTests/Write/FB_WriteRepeatedFieldFloatTests.TcPOU
FUNCTION_BLOCK INTERNAL FINAL FB_WriteRepeatedFieldFloatTests EXTENDS FB_TestSuite
VAR_INPUT
END_VAR
VAR_OUTPUT
END_VAR
VAR
	fbFieldCodec : FB_FieldCodecFloat(nTag:= 0);
	aActual    	 : ARRAY [0..7] OF REAL;
	fbRepeatedField		: FB_RepeatedField(anyArray:= F_ToAnyType(aActual), anyFirstElem:= F_ToAnyType(aActual[0]), ipFieldCodec:= fbFieldCodec);
END_VAR
(*
syntax = "proto3";

message MessageRepeatedFloat
{
  repeated float repeatedFloat = 4;
}


JSON:
{
  "repeatedFloat": [
    0, 1234.567, 1337.1337, -1.0, 12345678.321, 2147483647.65432
  ]
}

*)

ShouldWriteRepeatedFieldTheory();

METHOD PRIVATE Reset
VAR_INPUT
END_VAR
fbRepeatedField.Initialize();
MEMSET(destAddr:= ADR(aActual), fillByte:= 16#0, n:= SIZEOF(aActual));
END_METHOD

METHOD PRIVATE ShouldWriteRepeatedField
VAR_IN_OUT CONSTANT
    aExpected   : ARRAY [*] OF BYTE;
END_VAR
VAR_INPUT
    aValues     : ARRAY [0..7] OF REAL;
    nLength     : UDINT;
    nTag        : UDINT;
    nBufferPosStart     : UDINT;
    nExpectedBufferPos  : UDINT;
    ipFieldCodec        : I_FieldCodec;
END_VAR
VAR_INST
    fbCtx   : FB_WriteContext;
END_VAR
VAR
    aActualBuffer       : ARRAY [0..63] OF BYTE;
    hr                  : HRESULT;

END_VAR
// Arrange
Reset();
fbCtx.FromBuffer(aActualBuffer);
fbCtx.refCtx.stState.nBufferPos := nBufferPosStart;
ipFieldCodec.Tag := nTag;
fbRepeatedField.InitializeFromArray(anyArray:= F_ToAnyType(aValues), anyFirstElem:= F_ToAnyType(aValues[0]), nCount:= nLength);

// Act
hr := fbRepeatedField.WriteTo(fbWriteCtx:= fbCtx, ipFieldCodec:= ipFieldCodec);

// Assert
AssertEquals_DINT(
    Expected:= S_OK,
    Actual:= hr,
    Message:= 'Expected S_OK instead of error');
    
{warning disable C0041}
AssertArrayEquals_BYTE(Expecteds:= aExpected, Actuals:= aActualBuffer, Message:= '');
 
AssertEquals_UDINT(
    Expected:= nExpectedBufferPos,
    Actual:= fbCtx.refCtx.stState.nBufferPos,
    Message:= CONCAT('Expected stState.nBufferPos to equal ', TO_STRING(nExpectedBufferPos)));
END_METHOD

METHOD PRIVATE ShouldWriteRepeatedFieldTheory : REFERENCE TO FB_Test
VAR CONSTANT
    cRawValueZeroLength     : ARRAY[0..63] OF BYTE := [16#00, 16#00];
    cRawValue1              : ARRAY[0..63] OF BYTE := [16#00, 16#22, 16#18, 16#00, 16#00, 16#00, 16#00, 16#25, 16#52, 16#9a, 16#44, 16#47, 16#24, 16#a7, 16#44, 16#00, 16#00, 16#80, 16#bf, 16#4e, 16#61, 16#3c, 16#4b, 16#00, 16#00, 16#00, 16#4f];  
END_VAR

VAR CONSTANT
    aExpectedZeroLength     : ARRAY [0..7] OF REAL := [0, 0, 0, 0, 0, 0, 0, 0];
    aExpected1              : ARRAY [0..7] OF REAL := [0, 1234.567, 1337.1337, -1.0, 12345678.321, 2147483647.65432];
END_VAR
TEST(__POUNAME());

ShouldWriteRepeatedField(aExpected:= cRawValueZeroLength, aValues:= aExpectedZeroLength, nLength:= 0, nTag:= F_MakeTag(1, E_WireType.LengthDelimited), nBufferPosStart:= 0, nExpectedBufferPos:= 0, ipFieldCodec:= THIS^.fbFieldCodec);
ShouldWriteRepeatedField(aExpected:= cRawValue1, aValues:= aExpected1, nLength:= 6, nTag:= F_MakeTag(4, E_WireType.LengthDelimited), nBufferPosStart:= 1, nExpectedBufferPos:= 27, ipFieldCodec:= THIS^.fbFieldCodec);

TEST_FINISHED_NAMED(__POUNAME());
END_METHOD

END_FUNCTION_BLOCK

// ---- __TESTs/RepeatedFieldTests/Write/FB_WriteRepeatedFieldInt32Tests.TcPOU
FUNCTION_BLOCK INTERNAL FINAL FB_WriteRepeatedFieldInt32Tests EXTENDS FB_TestSuite
VAR_INPUT
END_VAR
VAR_OUTPUT
END_VAR
VAR
	fbFieldCodec : FB_FieldCodecInt32(nTag:= 0);
	aActual    	 : ARRAY [0..7] OF DINT;
	fbRepeatedField		: FB_RepeatedField(anyArray:= F_ToAnyType(aActual), anyFirstElem:= F_ToAnyType(aActual[0]), ipFieldCodec:= fbFieldCodec);
END_VAR

ShouldWriteRepeatedFieldTheory();

METHOD PRIVATE Reset
VAR_INPUT
END_VAR
fbRepeatedField.Initialize();
MEMSET(destAddr:= ADR(aActual), fillByte:= 16#0, n:= SIZEOF(aActual));
END_METHOD

METHOD PRIVATE ShouldWriteRepeatedField
VAR_IN_OUT CONSTANT
    aExpected   : ARRAY [*] OF BYTE;
END_VAR
VAR_INPUT
    aValues     : ARRAY [0..7] OF DINT;
    nLength     : UDINT;
    nTag        : UDINT;
    nBufferPosStart     : UDINT;
    nExpectedBufferPos  : UDINT;
    ipFieldCodec        : I_FieldCodec;
END_VAR
VAR_INST
    fbCtx   : FB_WriteContext;
END_VAR
VAR
    aActualBuffer       : ARRAY [0..63] OF BYTE;
    hr                  : HRESULT;

END_VAR
// Arrange
Reset();
fbCtx.FromBuffer(aActualBuffer);
fbCtx.refCtx.stState.nBufferPos := nBufferPosStart;
ipFieldCodec.Tag := nTag;
fbRepeatedField.InitializeFromArray(anyArray:= F_ToAnyType(aValues), anyFirstElem:= F_ToAnyType(aValues[0]), nCount:= nLength);

// Act
hr := fbRepeatedField.WriteTo(fbWriteCtx:= fbCtx, ipFieldCodec:= ipFieldCodec);

// Assert
AssertEquals_DINT(
    Expected:= S_OK,
    Actual:= hr,
    Message:= 'Expected S_OK instead of error');
    
{warning disable C0041}
AssertArrayEquals_BYTE(Expecteds:= aExpected, Actuals:= aActualBuffer, Message:= '');
 
AssertEquals_UDINT(
    Expected:= nExpectedBufferPos,
    Actual:= fbCtx.refCtx.stState.nBufferPos,
    Message:= CONCAT('Expected stState.nBufferPos to equal ', TO_STRING(nExpectedBufferPos)));
END_METHOD

METHOD PRIVATE ShouldWriteRepeatedFieldTheory : REFERENCE TO FB_Test
VAR CONSTANT
    cRawValueZeroLength     : ARRAY[0..63] OF BYTE := [16#00, 16#00];
    cRawValue1              : ARRAY[0..63] OF BYTE := [16#00, 16#0A, 16#18, 16#00, 16#D2, 16#09, 16#B9, 16#0A, 16#FF, 16#FF, 16#FF, 16#FF, 16#FF, 16#FF, 16#FF, 16#FF, 16#FF, 16#01, 16#CE, 16#C2, 16#F1, 16#05, 16#FF, 16#FF, 16#FF, 16#FF, 16#07];  
END_VAR

VAR CONSTANT
    aExpectedZeroLength     : ARRAY [0..7] OF DINT := [0, 0, 0, 0, 0, 0, 0, 0];
    aExpected1              : ARRAY [0..7] OF DINT := [0, 1234, 1337, -1, 12345678, 2147483647];
END_VAR
TEST(__POUNAME());

ShouldWriteRepeatedField(aExpected:= cRawValueZeroLength, aValues:= aExpectedZeroLength, nLength:= 0, nTag:= F_MakeTag(1, E_WireType.LengthDelimited), nBufferPosStart:= 0, nExpectedBufferPos:= 0, ipFieldCodec:= THIS^.fbFieldCodec);
ShouldWriteRepeatedField(aExpected:= cRawValue1, aValues:= aExpected1, nLength:= 6, nTag:= F_MakeTag(1, E_WireType.LengthDelimited), nBufferPosStart:= 1, nExpectedBufferPos:= 27, ipFieldCodec:= THIS^.fbFieldCodec);

TEST_FINISHED_NAMED(__POUNAME());
END_METHOD

END_FUNCTION_BLOCK

// ---- __TESTs/RepeatedFieldTests/Write/FB_WriteRepeatedFieldInt64Tests.TcPOU
FUNCTION_BLOCK INTERNAL FINAL FB_WriteRepeatedFieldInt64Tests EXTENDS FB_TestSuite
VAR_INPUT
END_VAR
VAR_OUTPUT
END_VAR
VAR
	fbFieldCodec : FB_FieldCodecInt64(nTag:= 0);
	aActual    	 : ARRAY [0..7] OF LINT;
	fbRepeatedField		: FB_RepeatedField(anyArray:= F_ToAnyType(aActual), anyFirstElem:= F_ToAnyType(aActual[0]), ipFieldCodec:= fbFieldCodec);
END_VAR

ShouldWriteRepeatedFieldTheory();

METHOD PRIVATE Reset
VAR_INPUT
END_VAR
fbRepeatedField.Initialize();
MEMSET(destAddr:= ADR(aActual), fillByte:= 16#0, n:= SIZEOF(aActual));
END_METHOD

METHOD PRIVATE ShouldWriteRepeatedField
VAR_IN_OUT CONSTANT
    aExpected   : ARRAY [*] OF BYTE;
END_VAR
VAR_INPUT
    aValues     : ARRAY [0..7] OF LINT;
    nLength     : UDINT;
    nTag        : UDINT;
    nBufferPosStart     : UDINT;
    nExpectedBufferPos  : UDINT;
    ipFieldCodec        : I_FieldCodec;
END_VAR
VAR_INST
    fbCtx   : FB_WriteContext;
END_VAR
VAR
    aActualBuffer       : ARRAY [0..63] OF BYTE;
    hr                  : HRESULT;
END_VAR
// Arrange
Reset();
fbCtx.FromBuffer(aActualBuffer);
fbCtx.refCtx.stState.nBufferPos := nBufferPosStart;
ipFieldCodec.Tag := nTag;
fbRepeatedField.InitializeFromArray(anyArray:= F_ToAnyType(aValues), anyFirstElem:= F_ToAnyType(aValues[0]), nCount:= nLength);

// Act
hr := fbRepeatedField.WriteTo(fbWriteCtx:= fbCtx, ipFieldCodec:= ipFieldCodec);

// Assert
AssertEquals_DINT(
    Expected:= S_OK,
    Actual:= hr,
    Message:= 'Expected S_OK instead of error');
    
{warning disable C0041}
AssertArrayEquals_BYTE(Expecteds:= aExpected, Actuals:= aActualBuffer, Message:= '');
 
AssertEquals_UDINT(
    Expected:= nExpectedBufferPos,
    Actual:= fbCtx.refCtx.stState.nBufferPos,
    Message:= CONCAT('Expected stState.nBufferPos to equal ', TO_STRING(nExpectedBufferPos)));
END_METHOD

METHOD PRIVATE ShouldWriteRepeatedFieldTheory : REFERENCE TO FB_Test
VAR CONSTANT
    cRawValueZeroLength     : ARRAY[0..63] OF BYTE := [16#00, 16#00];
    cRawValue1              : ARRAY[0..63] OF BYTE := [16#00, 16#0A, 16#18, 16#00, 16#D2, 16#09, 16#B9, 16#0A, 16#FF, 16#FF, 16#FF, 16#FF, 16#FF, 16#FF, 16#FF, 16#FF, 16#FF, 16#01, 16#CE, 16#C2, 16#F1, 16#05, 16#B4, 16#80, 16#80, 16#80, 16#08];  
END_VAR

VAR CONSTANT
    aExpectedZeroLength     : ARRAY [0..7] OF LINT := [0, 0, 0, 0, 0, 0, 0, 0];
    aExpected1              : ARRAY [0..7] OF LINT := [0, 1234, 1337, -1, 12345678, 2147483700];
END_VAR
TEST(__POUNAME());

ShouldWriteRepeatedField(aExpected:= cRawValueZeroLength, aValues:= aExpectedZeroLength, nLength:= 0, nTag:= F_MakeTag(1, E_WireType.LengthDelimited), nBufferPosStart:= 0, nExpectedBufferPos:= 0, ipFieldCodec:= THIS^.fbFieldCodec);
ShouldWriteRepeatedField(aExpected:= cRawValue1, aValues:= aExpected1, nLength:= 6, nTag:= F_MakeTag(1, E_WireType.LengthDelimited), nBufferPosStart:= 1, nExpectedBufferPos:= 27, ipFieldCodec:= THIS^.fbFieldCodec);

TEST_FINISHED_NAMED(__POUNAME());
END_METHOD

END_FUNCTION_BLOCK

// ---- __TESTs/RepeatedFieldTests/Write/FB_WriteRepeatedFieldMessageTests.TcPOU
FUNCTION_BLOCK INTERNAL FB_WriteRepeatedFieldMessageTests EXTENDS FB_TestSuite
VAR
	fbWriteCtx		: FB_WriteContext;
	fbFoo   		: FB_Foo;
	stFoo           : ST_Foo;
	aBuffer 		: ARRAY[0..255] OF BYTE;
END_VAR

TEST(__POUNAME());


// Arrange
fbWriteCtx.FromBuffer(aBuffer);
stFoo.baz[0].value:= 42;
stFoo.baz[0].name:= 'foo';
stFoo.baz[1].value:= 6969;
stFoo.baz[1].name:= 'bar';
stFoo.baz[2].value:= 1337;
stFoo.baz[2].name:= 'baz';
F_SetMessageValue(F_ToAnyType(stFoo), fbFoo);

// Act 
fbFoo.WriteTo(fbWriteCtx);



// Assert



TEST_FINISHED_NAMED(__POUNAME());

END_FUNCTION_BLOCK

// ---- __TESTs/RepeatedFieldTests/Write/FB_WriteRepeatedFieldSInt32Tests.TcPOU
FUNCTION_BLOCK INTERNAL FINAL FB_WriteRepeatedFieldSInt32Tests EXTENDS FB_TestSuite
VAR_INPUT
END_VAR
VAR_OUTPUT
END_VAR
VAR
	fbFieldCodec : FB_FieldCodecSInt32(nTag:= 0);
	aActual    	 : ARRAY [0..7] OF DINT;
	fbRepeatedField		: FB_RepeatedField(anyArray:= F_ToAnyType(aActual), anyFirstElem:= F_ToAnyType(aActual[0]), ipFieldCodec:= fbFieldCodec);
END_VAR

ShouldWriteRepeatedFieldTheory();

METHOD PRIVATE Reset
VAR_INPUT
END_VAR
fbRepeatedField.Initialize();
MEMSET(destAddr:= ADR(aActual), fillByte:= 16#0, n:= SIZEOF(aActual));
END_METHOD

METHOD PRIVATE ShouldWriteRepeatedField
VAR_IN_OUT CONSTANT
    aExpected   : ARRAY [*] OF BYTE;
END_VAR
VAR_INPUT
    aValues     : ARRAY [0..7] OF DINT;
    nLength     : UDINT;
    nTag        : UDINT;
    nBufferPosStart     : UDINT;
    nExpectedBufferPos  : UDINT;
    ipFieldCodec        : I_FieldCodec;
END_VAR
VAR_INST
    fbCtx   : FB_WriteContext;
END_VAR
VAR
    aActualBuffer       : ARRAY [0..63] OF BYTE;
    hr                  : HRESULT;

END_VAR
// Arrange
Reset();
fbCtx.FromBuffer(aActualBuffer);
fbCtx.refCtx.stState.nBufferPos := nBufferPosStart;
ipFieldCodec.Tag := nTag;
fbRepeatedField.InitializeFromArray(anyArray:= F_ToAnyType(aValues), anyFirstElem:= F_ToAnyType(aValues[0]), nCount:= nLength);

// Act
hr := fbRepeatedField.WriteTo(fbWriteCtx:= fbCtx, ipFieldCodec:= ipFieldCodec);

// Assert
AssertEquals_DINT(
    Expected:= S_OK,
    Actual:= hr,
    Message:= 'Expected S_OK instead of error');
    
{warning disable C0041}
AssertArrayEquals_BYTE(Expecteds:= aExpected, Actuals:= aActualBuffer, Message:= '');
 
AssertEquals_UDINT(
    Expected:= nExpectedBufferPos,
    Actual:= fbCtx.refCtx.stState.nBufferPos,
    Message:= CONCAT('Expected stState.nBufferPos to equal ', TO_STRING(nExpectedBufferPos)));
END_METHOD

METHOD PRIVATE ShouldWriteRepeatedFieldTheory : REFERENCE TO FB_Test
VAR CONSTANT
    cRawValueZeroLength     : ARRAY[0..63] OF BYTE := [16#00, 16#00];
    cRawValue1              : ARRAY[0..63] OF BYTE := [16#00, 16#0A, 16#09, 16#00, 16#02, 16#01, 16#F2, 16#14, 16#F1, 16#14, 16#F2, 16#6C];  
END_VAR

VAR CONSTANT
    aExpectedZeroLength     : ARRAY [0..7] OF DINT := [0, 0, 0, 0, 0, 0, 0, 0];
    aExpected1              : ARRAY [0..7] OF DINT := [0, 1, -1, 1337, -1337, 6969, 0];
END_VAR
TEST(__POUNAME());

ShouldWriteRepeatedField(aExpected:= cRawValueZeroLength, aValues:= aExpectedZeroLength, nLength:= 0, nTag:= F_MakeTag(1, E_WireType.LengthDelimited), nBufferPosStart:= 0, nExpectedBufferPos:= 0, ipFieldCodec:= THIS^.fbFieldCodec);
ShouldWriteRepeatedField(aExpected:= cRawValue1, aValues:= aExpected1, nLength:= 6, nTag:= F_MakeTag(1, E_WireType.LengthDelimited), nBufferPosStart:= 1, nExpectedBufferPos:= 12, ipFieldCodec:= THIS^.fbFieldCodec);

TEST_FINISHED_NAMED(__POUNAME());
END_METHOD

END_FUNCTION_BLOCK

// ---- __TESTs/RepeatedFieldTests/Write/FB_WriteRepeatedFieldSInt64Tests.TcPOU
FUNCTION_BLOCK INTERNAL FINAL FB_WriteRepeatedFieldSInt64Tests EXTENDS FB_TestSuite
VAR_INPUT
END_VAR
VAR_OUTPUT
END_VAR
VAR
	fbFieldCodec : FB_FieldCodecSInt64(nTag:= 0);
	aActual    	 : ARRAY [0..7] OF DINT;
	fbRepeatedField		: FB_RepeatedField(anyArray:= F_ToAnyType(aActual), anyFirstElem:= F_ToAnyType(aActual[0]), ipFieldCodec:= fbFieldCodec);
END_VAR

ShouldWriteRepeatedFieldTheory();

METHOD PRIVATE Reset
VAR_INPUT
END_VAR
fbRepeatedField.Initialize();
MEMSET(destAddr:= ADR(aActual), fillByte:= 16#0, n:= SIZEOF(aActual));
END_METHOD

METHOD PRIVATE ShouldWriteRepeatedField
VAR_IN_OUT CONSTANT
    aExpected   : ARRAY [*] OF BYTE;
END_VAR
VAR_INPUT
    aValues     : ARRAY [0..7] OF LINT;
    nLength     : UDINT;
    nTag        : UDINT;
    nBufferPosStart     : UDINT;
    nExpectedBufferPos  : UDINT;
    ipFieldCodec        : I_FieldCodec;
END_VAR
VAR_INST
    fbCtx   : FB_WriteContext;
END_VAR
VAR
    aActualBuffer       : ARRAY [0..63] OF BYTE;
    hr                  : HRESULT;

END_VAR
// Arrange
Reset();
fbCtx.FromBuffer(aActualBuffer);
fbCtx.refCtx.stState.nBufferPos := nBufferPosStart;
ipFieldCodec.Tag := nTag;
fbRepeatedField.InitializeFromArray(anyArray:= F_ToAnyType(aValues), anyFirstElem:= F_ToAnyType(aValues[0]), nCount:= nLength);

// Act
hr := fbRepeatedField.WriteTo(fbWriteCtx:= fbCtx, ipFieldCodec:= ipFieldCodec);

// Assert
AssertEquals_DINT(
    Expected:= S_OK,
    Actual:= hr,
    Message:= 'Expected S_OK instead of error');
    
{warning disable C0041}
AssertArrayEquals_BYTE(Expecteds:= aExpected, Actuals:= aActualBuffer, Message:= '');
 
AssertEquals_UDINT(
    Expected:= nExpectedBufferPos,
    Actual:= fbCtx.refCtx.stState.nBufferPos,
    Message:= CONCAT('Expected stState.nBufferPos to equal ', TO_STRING(nExpectedBufferPos)));
END_METHOD

METHOD PRIVATE ShouldWriteRepeatedFieldTheory : REFERENCE TO FB_Test
VAR CONSTANT
    cRawValueZeroLength     : ARRAY[0..63] OF BYTE := [16#00, 16#00];
    cRawValue1              : ARRAY[0..63] OF BYTE := [16#00, 16#0A, 16#11, 16#00, 16#A4, 16#13, 16#F2, 16#14, 16#01, 16#F1, 16#14, 16#9C, 16#85, 16#E3, 16#0B, 16#E7, 16#80, 16#80, 16#80, 16#10];  
END_VAR

VAR CONSTANT
    aExpectedZeroLength     : ARRAY [0..7] OF LINT := [0, 0, 0, 0, 0, 0, 0, 0];
    aExpected1              : ARRAY [0..7] OF LINT := [0, 1234, 1337, -1, -1337, 12345678, -2147483700, 0];
END_VAR
TEST(__POUNAME());

ShouldWriteRepeatedField(aExpected:= cRawValueZeroLength, aValues:= aExpectedZeroLength, nLength:= 0, nTag:= F_MakeTag(1, E_WireType.LengthDelimited), nBufferPosStart:= 0, nExpectedBufferPos:= 0, ipFieldCodec:= THIS^.fbFieldCodec);
ShouldWriteRepeatedField(aExpected:= cRawValue1, aValues:= aExpected1, nLength:= 7, nTag:= F_MakeTag(1, E_WireType.LengthDelimited), nBufferPosStart:= 1, nExpectedBufferPos:= 20, ipFieldCodec:= THIS^.fbFieldCodec);

TEST_FINISHED_NAMED(__POUNAME());
END_METHOD

END_FUNCTION_BLOCK

// ---- __TESTs/RepeatedFieldTests/Write/FB_WriteRepeatedFieldStringTests.TcPOU
FUNCTION_BLOCK INTERNAL FINAL FB_WriteRepeatedFieldStringTests EXTENDS FB_TestSuite
VAR_INPUT
END_VAR
VAR_OUTPUT
END_VAR
VAR
    fbFieldCodec : FB_FieldCodecString(nTag:= 0);
	aActual     : ARRAY [0..15] OF T_MAXSTRING;
	fbRepeatedField		: FB_RepeatedField(anyArray:= F_ToAnyType(aActual), anyFirstElem:= F_ToAnyType(aActual[0]), ipFieldCodec:= fbFieldCodec);
END_VAR

ShouldWriteRepeatedFieldTheory();

METHOD PRIVATE Reset
VAR_INPUT
END_VAR
fbRepeatedField.Initialize();
MEMSET(destAddr:= ADR(aActual), fillByte:= 16#0, n:= SIZEOF(aActual));
END_METHOD

METHOD PRIVATE ShouldWriteRepeatedField
VAR_IN_OUT CONSTANT
    aExpected   : ARRAY [*] OF BYTE;
END_VAR
VAR_INPUT
    aValues     : ARRAY [0..15] OF T_MAXSTRING;
    nLength     : UDINT;
    nTag        : UDINT;
    nBufferPosStart     : UDINT;
    nExpectedBufferPos  : UDINT;
    ipFieldCodec        : I_FieldCodec;
END_VAR
VAR_INST
    fbCtx   : FB_WriteContext;
END_VAR
VAR
    aActualBuffer       : ARRAY [0..255] OF BYTE;
    hr                  : HRESULT;
END_VAR
// Arrange
Reset();
fbCtx.FromBuffer(aActualBuffer);
fbCtx.refCtx.stState.nBufferPos := nBufferPosStart;
ipFieldCodec.Tag := nTag;
fbRepeatedField.InitializeFromArray(anyArray:= F_ToAnyType(aValues), anyFirstElem:= F_ToAnyType(aValues[0]), nCount:= nLength);

// Act
hr := fbRepeatedField.WriteTo(fbWriteCtx:= fbCtx, ipFieldCodec:= ipFieldCodec);

// Assert
AssertEquals_DINT(
    Expected:= S_OK,
    Actual:= hr,
    Message:= 'Expected S_OK instead of error');
    
{warning disable C0041}
AssertArrayEquals_BYTE(Expecteds:= aExpected, Actuals:= aActualBuffer, Message:= '');
 
AssertEquals_UDINT(
    Expected:= nExpectedBufferPos,
    Actual:= fbCtx.refCtx.stState.nBufferPos,
    Message:= CONCAT('Expected stState.nBufferPos to equal ', TO_STRING(nExpectedBufferPos)));
END_METHOD

METHOD PRIVATE ShouldWriteRepeatedFieldTheory : REFERENCE TO FB_Test
VAR CONSTANT
    aExpectedBufferZeroLen  : ARRAY[0..255] OF BYTE := [16#00, 16#00];
    aExpectedBuffer1        : ARRAY[0..255] OF BYTE := [16#0A, 16#0B, 16#54, 16#65, 16#73, 16#74, 16#53, 16#74, 16#72, 16#69, 16#6E, 16#67, 16#30, 16#0A, 16#0B, 16#54, 16#65, 16#73, 16#74, 16#53, 16#74, 16#72, 16#69, 16#6E, 16#67, 16#31, 16#0A, 16#0B, 16#54, 16#65, 16#73, 16#74, 16#53, 16#74, 16#72, 16#69, 16#6E, 16#67, 16#32, 16#0A, 16#0B, 16#54, 16#65, 16#73, 16#74, 16#53, 16#74, 16#72, 16#69, 16#6E, 16#67, 16#33];
    aExpectedBuffer2        : ARRAY[0..255] OF BYTE := [16#00, 16#0A, 16#28, 16#75, 16#74, 16#66, 16#2D, 16#38, 16#3A, 16#20, 16#61, 16#2D, 16#7A, 16#2C, 16#20, 16#41, 16#2D, 16#5A, 16#2C, 16#20, 16#30, 16#2D, 16#39, 16#2C, 16#20, 16#C3, 16#A4, 16#C3, 16#84, 16#C3, 16#B6, 16#C3, 16#96, 16#C3, 16#BC, 16#C3, 16#9C, 16#C3, 16#9F, 16#F0, 16#9F, 16#9A, 16#80, 16#0A, 16#06, 16#30, 16#31, 16#32, 16#33, 16#34, 16#35];
END_VAR

VAR CONSTANT
    aValueZeroLen           : ARRAY[0..15] OF T_MAXSTRING := [];
    aValue1                 : ARRAY[0..15] OF T_MAXSTRING := ['TestString0', 'TestString1', 'TestString2', 'TestString3'];
    aValue2                 : ARRAY[0..15] OF T_MAXSTRING := ['utf-8: a-z, A-Z, 0-9, äÄöÖüÜß🚀', '012345'];
END_VAR
TEST(__POUNAME());
ShouldWriteRepeatedField(aExpected:= aExpectedBufferZeroLen, aValues:= aValueZeroLen, nLength:= 0, nTag:= F_MakeTag(1, E_WireType.LengthDelimited), nBufferPosStart:= 0, nExpectedBufferPos:= 0, ipFieldCodec:= THIS^.fbFieldCodec);
ShouldWriteRepeatedField(aExpected:= aExpectedBuffer1, aValues:= aValue1, nLength:= 4, nTag:= F_MakeTag(1, E_WireType.LengthDelimited), nBufferPosStart:= 0, nExpectedBufferPos:= 52, ipFieldCodec:= THIS^.fbFieldCodec);
ShouldWriteRepeatedField(aExpected:= aExpectedBuffer2, aValues:= aValue2, nLength:= 2, nTag:= F_MakeTag(1, E_WireType.LengthDelimited), nBufferPosStart:= 1, nExpectedBufferPos:= 51, ipFieldCodec:= THIS^.fbFieldCodec);
TEST_FINISHED_NAMED(__POUNAME());
END_METHOD

END_FUNCTION_BLOCK

// ---- __TESTs/RepeatedFieldTests/Write/FB_WriteRepeatedFieldUint32Tests.TcPOU
FUNCTION_BLOCK INTERNAL FINAL FB_WriteRepeatedFieldUint32Tests EXTENDS FB_TestSuite
VAR_INPUT
END_VAR
VAR_OUTPUT
END_VAR
VAR
	fbFieldCodec : FB_FieldCodecUInt32(nTag:= 0);
	aActual    	 : ARRAY [0..7] OF UDINT;
	fbRepeatedField		: FB_RepeatedField(anyArray:= F_ToAnyType(aActual), anyFirstElem:= F_ToAnyType(aActual[0]), ipFieldCodec:= fbFieldCodec);
END_VAR

ShouldWriteRepeatedFieldTheory();

METHOD PRIVATE Reset
VAR_INPUT
END_VAR
fbRepeatedField.Initialize();
MEMSET(destAddr:= ADR(aActual), fillByte:= 16#0, n:= SIZEOF(aActual));
END_METHOD

METHOD PRIVATE ShouldWriteRepeatedField
VAR_IN_OUT CONSTANT
    aExpected   : ARRAY [*] OF BYTE;
END_VAR
VAR_INPUT
    aValues     : ARRAY [0..7] OF UDINT;
    nLength     : UDINT;
    nTag        : UDINT;
    nBufferPosStart     : UDINT;
    nExpectedBufferPos  : UDINT;
    ipFieldCodec        : I_FieldCodec;
END_VAR
VAR_INST
    fbCtx   : FB_WriteContext;
END_VAR
VAR
    aActualBuffer       : ARRAY [0..63] OF BYTE;
    hr                  : HRESULT;

END_VAR
// Arrange
Reset();
fbCtx.FromBuffer(aActualBuffer);
fbCtx.refCtx.stState.nBufferPos := nBufferPosStart;
ipFieldCodec.Tag := nTag;
fbRepeatedField.InitializeFromArray(anyArray:= F_ToAnyType(aValues), anyFirstElem:= F_ToAnyType(aValues[0]), nCount:= nLength);

// Act
hr := fbRepeatedField.WriteTo(fbWriteCtx:= fbCtx, ipFieldCodec:= ipFieldCodec);

// Assert
AssertEquals_DINT(
    Expected:= S_OK,
    Actual:= hr,
    Message:= 'Expected S_OK instead of error');
    
{warning disable C0041}
AssertArrayEquals_BYTE(Expecteds:= aExpected, Actuals:= aActualBuffer, Message:= '');
 
AssertEquals_UDINT(
    Expected:= nExpectedBufferPos,
    Actual:= fbCtx.refCtx.stState.nBufferPos,
    Message:= CONCAT('Expected stState.nBufferPos to equal ', TO_STRING(nExpectedBufferPos)));
END_METHOD

METHOD PRIVATE ShouldWriteRepeatedFieldTheory : REFERENCE TO FB_Test
VAR CONSTANT
    cRawValueZeroLength     : ARRAY[0..63] OF BYTE := [16#00, 16#00];
    cRawValue1              : ARRAY[0..63] OF BYTE := [16#00, 16#0A, 16#07, 16#00, 16#01, 16#FF, 16#01, 16#96, 16#01, 16#04];  
END_VAR

VAR CONSTANT
    aExpectedZeroLength     : ARRAY [0..7] OF UDINT := [0, 0, 0, 0, 0, 0, 0, 0];
    aExpected1              : ARRAY [0..7] OF UDINT := [0, 1, 255, 150, 4, 0, 0, 0];
END_VAR
TEST(__POUNAME());

ShouldWriteRepeatedField(aExpected:= cRawValueZeroLength, aValues:= aExpectedZeroLength, nLength:= 0, nTag:= F_MakeTag(1, E_WireType.LengthDelimited), nBufferPosStart:= 0, nExpectedBufferPos:= 0, ipFieldCodec:= THIS^.fbFieldCodec);
ShouldWriteRepeatedField(aExpected:= cRawValue1, aValues:= aExpected1, nLength:= 5, nTag:= F_MakeTag(1, E_WireType.LengthDelimited), nBufferPosStart:= 1, nExpectedBufferPos:= 10, ipFieldCodec:= THIS^.fbFieldCodec);

TEST_FINISHED_NAMED(__POUNAME());
END_METHOD

END_FUNCTION_BLOCK

// ---- __TESTs/RepeatedFieldTests/Write/FB_WriteRepeatedFieldUint64Tests.TcPOU
FUNCTION_BLOCK INTERNAL FINAL FB_WriteRepeatedFieldUint64Tests EXTENDS FB_TestSuite
VAR_INPUT
END_VAR
VAR_OUTPUT
END_VAR
VAR
	fbFieldCodec : FB_FieldCodecUInt64(nTag:= 0);
	aActual    	 : ARRAY [0..7] OF ULINT;
	fbRepeatedField		: FB_RepeatedField(anyArray:= F_ToAnyType(aActual), anyFirstElem:= F_ToAnyType(aActual[0]), ipFieldCodec:= fbFieldCodec);
END_VAR

ShouldWriteRepeatedFieldTheory();

METHOD PRIVATE Reset
VAR_INPUT
END_VAR
fbRepeatedField.Initialize();
MEMSET(destAddr:= ADR(aActual), fillByte:= 16#0, n:= SIZEOF(aActual));
END_METHOD

METHOD PRIVATE ShouldWriteRepeatedField
VAR_IN_OUT CONSTANT
    aExpected   : ARRAY [*] OF BYTE;
END_VAR
VAR_INPUT
    aValues     : ARRAY [0..7] OF ULINT;
    nLength     : UDINT;
    nTag        : UDINT;
    nBufferPosStart     : UDINT;
    nExpectedBufferPos  : UDINT;
    ipFieldCodec        : I_FieldCodec;
END_VAR
VAR_INST
    fbCtx   : FB_WriteContext;
END_VAR
VAR
    aActualBuffer       : ARRAY [0..63] OF BYTE;
    hr                  : HRESULT;

END_VAR
// Arrange
Reset();
fbCtx.FromBuffer(aActualBuffer);
fbCtx.refCtx.stState.nBufferPos := nBufferPosStart;
ipFieldCodec.Tag := nTag;
fbRepeatedField.InitializeFromArray(anyArray:= F_ToAnyType(aValues), anyFirstElem:= F_ToAnyType(aValues[0]), nCount:= nLength);

// Act
hr := fbRepeatedField.WriteTo(fbWriteCtx:= fbCtx, ipFieldCodec:= ipFieldCodec);

// Assert
AssertEquals_DINT(
    Expected:= S_OK,
    Actual:= hr,
    Message:= 'Expected S_OK instead of error');
    
{warning disable C0041}
AssertArrayEquals_BYTE(Expecteds:= aExpected, Actuals:= aActualBuffer, Message:= '');
 
AssertEquals_UDINT(
    Expected:= nExpectedBufferPos,
    Actual:= fbCtx.refCtx.stState.nBufferPos,
    Message:= CONCAT('Expected stState.nBufferPos to equal ', TO_STRING(nExpectedBufferPos)));
END_METHOD

METHOD PRIVATE ShouldWriteRepeatedFieldTheory : REFERENCE TO FB_Test
VAR CONSTANT
    cRawValueZeroLength     : ARRAY[0..63] OF BYTE := [16#00, 16#00];
    cRawValue1              : ARRAY[0..63] OF BYTE := [16#00, 16#0A, 16#0F, 16#00, 16#2A, 16#D2, 16#09, 16#B9, 16#0A, 16#95, 16#9A, 16#EF, 16#3A, 16#B4, 16#80, 16#80, 16#80, 16#08];  
END_VAR

VAR CONSTANT
    aExpectedZeroLength     : ARRAY [0..7] OF ULINT := [0, 0, 0, 0, 0, 0, 0, 0];
    aExpected1              : ARRAY [0..7] OF ULINT := [0, 42, 1234, 1337, 123456789, 2147483700, 0];
END_VAR
TEST(__POUNAME());

ShouldWriteRepeatedField(aExpected:= cRawValueZeroLength, aValues:= aExpectedZeroLength, nLength:= 0, nTag:= F_MakeTag(1, E_WireType.LengthDelimited), nBufferPosStart:= 0, nExpectedBufferPos:= 0, ipFieldCodec:= THIS^.fbFieldCodec);
ShouldWriteRepeatedField(aExpected:= cRawValue1, aValues:= aExpected1, nLength:= 6, nTag:= F_MakeTag(1, E_WireType.LengthDelimited), nBufferPosStart:= 1, nExpectedBufferPos:= 18, ipFieldCodec:= THIS^.fbFieldCodec);

TEST_FINISHED_NAMED(__POUNAME());
END_METHOD

END_FUNCTION_BLOCK
